(* PLC project Ethercat.project, CODESYS CODESYS V3.5 SP20 Patch 1 *)
(* stored: creationDateTime 2024-07-03T17:40:48.9144031, modificationDateTime 2024-07-03T17:14:47.7302062 *)

PROGRAM PLC_PRG
  VAR
    Blink : TON;
    Blink2 : TON;
    Output1 : BOOL;
    Start1 : BOOL;
    Start2 : BOOL;
    Fin1 : BOOL;
    Fin2 : BOOL;
    Cyclestate : INT;
  END_VAR

                    Blink(IN:= Start1, PT:= T#1000MS, Q=> Fin1, ET=> );
Blink2(IN:= Start2, PT:= T#1000MS, Q=> Fin2 , ET=> );
CASE Cyclestate OF	
	0:
		Start1 := TRUE;
		Output1 := TRUE;		
		Fin2 := FALSE;
		Cyclestate := 10;		
	10:
		IF Fin1 THEN
			Start1 := FALSE;
			Output1 := FALSE;			
			Cyclestate := 20;
		ELSE
			Cyclestate := 10;
		END_IF		
	20:
		Start2 := TRUE;
		Cyclestate := 30;
		Fin1 := FALSE;		
	30:
		IF Fin2 THEN
			Start2 := FALSE;
			Cyclestate := 0;
		ELSE
			Cyclestate := 30;
		END_IF
END_CASE
                  
END_PROGRAM

CONFIGURATION Device
  RESOURCE Application ON PLC
    TASK MainTask(INTERVAL := T#4ms, PRIORITY := 1);
    TASK EtherCAT_Task(INTERVAL := T#4ms, PRIORITY := 1);
    PROGRAM PLC_PRG WITH MainTask : PLC_PRG;
  END_RESOURCE
END_CONFIGURATION

CONFIGURATION EtherCAT_Master
END_CONFIGURATION

CONFIGURATION EP6224_0002
END_CONFIGURATION

CONFIGURATION Digital_Output
END_CONFIGURATION

CONFIGURATION <Empty>
END_CONFIGURATION

CONFIGURATION <Empty>
END_CONFIGURATION

CONFIGURATION <Empty>
END_CONFIGURATION

CONFIGURATION GPIOs_A_B
END_CONFIGURATION
